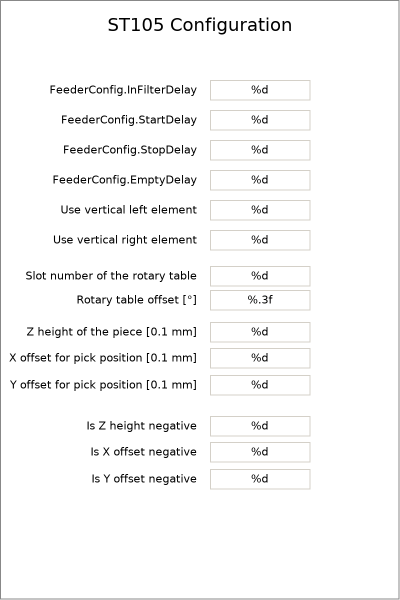
VISUALIZATION VISU_Recipe_ST105  // 400x600
    Textfield (210,80 100x20), "%d", text variable: _20_AUTO.recipe.st110.FeederConfig.InFilterDelay
        OnMouseDown: write the text variable via Default
    Label (0,5 400x40), "ST105 Configuration"
    Label (0,80 200x20), "FeederConfig.InFilterDelay"
    Textfield (210,110 100x20), "%d", text variable: _20_AUTO.recipe.st110.FeederConfig.StartDelay
        OnMouseDown: write the text variable via Default
    Label (0,110 200x20), "FeederConfig.StartDelay"
    Textfield (210,140 100x20), "%d", text variable: _20_AUTO.recipe.st105.FeederConfig.StopDelay
        OnMouseDown: write the text variable via Default
    Label (0,140 200x20), "FeederConfig.StopDelay"
    Textfield (210,170 100x20), "%d", text variable: _20_AUTO.recipe.st105.FeederConfig.EmptyDelay
        OnMouseDown: write the text variable via Default
    Label (0,170 200x20), "FeederConfig.EmptyDelay"
    Label (0,200 200x20), "Use vertical left element"
    Label (0,230 200x20), "Use vertical right element"
    Textfield (210,200 100x20), "%d", text variable: _20_AUTO.recipe.st105.xUseVerLeft
        OnMouseDown: write the text variable via Default
    Textfield (210,230 100x20), "%d", text variable: _20_AUTO.recipe.st105.xUseVerRight
        OnMouseDown: write the text variable via Default
    Textfield (210,416 100x20), "%d", text variable: _20_AUTO.recipe.st105.isPickUpPos_Z_neg
        OnMouseDown: write the text variable via Default
    Label (0,442 200x20), "Is X offset negative"
    Textfield (210,442 100x20), "%d", text variable: _20_AUTO.recipe.st105.isPickOffset_X_neg
        OnMouseDown: write the text variable via Default
    Label (0,469 200x20), "Is Y offset negative"
    Textfield (210,469 100x20), "%d", text variable: _20_AUTO.recipe.st105.isPickOffset_Y_neg
        OnMouseDown: write the text variable via Default
    Label (0,416 200x20), "Is Z height negative"
    Textfield (210,322 100x20), "%d", text variable: _20_AUTO.recipe.st105.PickUpPos_Z_deci
        OnMouseDown: write the text variable via Default
    Label (0,348 200x20), "X offset for pick position [0.1 mm]"
    Textfield (210,348 100x20), "%d", text variable: _20_AUTO.recipe.st105.PickOffset_X_deci
        OnMouseDown: write the text variable via Default
    Label (0,375 200x20), "Y offset for pick position [0.1 mm]"
    Textfield (210,375 100x20), "%d", text variable: _20_AUTO.recipe.st105.PickOffset_Y_deci
        OnMouseDown: write the text variable via Default
    Label (0,322 200x20), "Z height of the piece [0.1 mm]"
    Label (0,266 200x20), "Slot number of the rotary table"
    Textfield (210,266 100x20), "%d", text variable: _20_AUTO.recipe.st105.FeederSize
        OnMouseDown: write the text variable via Default
    Textfield (210,290 100x20), "%.3f", text variable: _20_AUTO.recipe.st105.RotaryTableOffset
        OnMouseDown: write the text variable via Default
    Label (0,290 200x20), "Rotary table offset [°]"
END_VISUALIZATION

(* stored: Version 1.1.0.1, ProductVersion 3.1.4024.6
   Visu VISU_Recipe_ST105: Id {8a5bb4e9-de39-4b81-a9d2-d23cd05df289} *)
